(*
Geographic Pose
----------------

Overview
================
Represents a coordinate system on a reference ellipsoid.
Similar to the HMatrix transformation, but based on an ellipsoid instead of in cartesian space (helper functions are included to switch between HMatrix and GeoPose).
Represents the geodetic (or geocentric) position with latitude, longitude, and elevation (above the ellipsoid) - Accessed with the 'Position' property.
Represents the orientation as a set of angles relative to the ENU tangent coordinate system at the CS origin - Accessed with the 'Orientation' property.
*)
FUNCTION_BLOCK GeoPose
VAR_INPUT
END_VAR
VAR_OUTPUT
END_VAR
VAR
	Position_ : GeoPosition;//ECEF
	Orientation_ : TaitBryanAngleOrientation;//ENU at position
END_VAR

METHOD PUBLIC Clear
VAR_INPUT
END_VAR
Position_.Clear();
Orientation_.Clear();
END_METHOD

METHOD PUBLIC CopyFrom
VAR_INPUT
	P : GeoPose;
END_VAR
Position_.CopyFrom(P.Position_);
Orientation_.CopyFrom(P.Orientation_);
END_METHOD

METHOD PUBLIC GetEcefTransformation : HMatrix
VAR_INPUT
	Ref : REFERENCE TO GeoEllipsoid := GeoEllipsoids.WGS84;
END_VAR
VAR
	EnuInEcef : HMatrix;//holds the geoposition part, and the tangent rotation
	ThisInEnu : HMatrix;//just holds the local rotation portion
END_VAR
EnuInEcef := Position_.GetTangentEnuTransform(Ref);
ThisInEnu.RMatrixComponent := Orientation_.GetRMatrix();
GetEcefTransformation := EnuInEcef.GetTransformedHMatrix(ThisInEnu);
END_METHOD

METHOD PUBLIC GetRelativeOrientation : TaitBryanAngleOrientation
VAR_INPUT
	P : GeoPose;
	Ref : REFERENCE TO GeoEllipsoid := GeoEllipsoids.WGS84;
END_VAR
VAR
	ThisInEcef : HMatrix;
	InputInThis : HMatrix;
END_VAR
ThisInEcef := GetEcefTransformation(Ref);
InputInThis := ThisInEcef.GetTransformedHMatrixReverse(P.GetEcefTransformation(Ref));
GetRelativeOrientation.SetFromRMatrix(InputInThis.RMatrixComponent);
END_METHOD

METHOD PUBLIC GetRelativePosition : Vector3
VAR_INPUT
	P : GeoPose;
	Ref : REFERENCE TO GeoEllipsoid := GeoEllipsoids.WGS84;
END_VAR
VAR
	ThisInEcef : HMatrix;
	InputInThis : HMatrix;
END_VAR
ThisInEcef := GetEcefTransformation(Ref);
InputInThis := ThisInEcef.GetTransformedHMatrixReverse(P.GetEcefTransformation(Ref));
GetRelativePosition := InputInThis.Vector3Component;
END_METHOD

METHOD PUBLIC IsEqual : BOOL
VAR_INPUT
	P : GeoPose;
END_VAR
IsEqual := IsNearlyEqual(P,0.0,0.0,0.0);
END_METHOD

METHOD PUBLIC IsNearlyEqual : BOOL
VAR_INPUT
	P : GeoPose;
	PositionPrecisionLatLon : LREAL;//rad
	PositionPrecisionElevation : LREAL;//m
	OrientationPrecision : LREAL;//radians
END_VAR
IsNearlyEqual := Position_.IsNearlyEqual(P.Position_, PositionPrecisionLatLon, PositionPrecisionElevation) AND Orientation_.IsNearlyEqual(P.Orientation_, OrientationPrecision);
END_METHOD

PROPERTY PUBLIC Orientation : TaitBryanAngleOrientation
GET
Orientation.CopyFrom(Orientation_);
END_GET
SET
Orientation_.CopyFrom(Orientation);
END_SET
END_PROPERTY

PROPERTY PUBLIC Position : GeoPosition
GET
Position.CopyFrom(Position_);
END_GET
SET
Position_.CopyFrom(Position);
END_SET
END_PROPERTY

METHOD PUBLIC SetFromComponents
VAR_INPUT
	P : GeoPosition;
	O : TaitBryanAngleOrientation;
END_VAR
Position_.CopyFrom(P);
Orientation_.CopyFrom(O);
END_METHOD

METHOD PUBLIC SetFromEcefTransformation
VAR_INPUT
	H : HMatrix;//ThisInEcef)
	Ref : REFERENCE TO GeoEllipsoid := GeoEllipsoids.WGS84;
END_VAR
VAR
	EnuInEcef : HMatrix;
	ThisInEnu : HMatrix;
END_VAR
Clear();
Position_.SetFromCartesianPosition(H.Vector3Component,Ref);
EnuInEcef := Position_.GetTangentEnuTransform(Ref);
ThisInEnu := EnuInEcef.GetTransformedHMatrixReverse(H);
Orientation_.SetFromRMatrix(ThisInEnu.RMatrixComponent);
END_METHOD

END_FUNCTION_BLOCK

(* stored: Version 1.1.0.1, ProductVersion 3.1.4024.9
   POU GeoPose: Id {22fd7b91-e379-4b48-b25b-7c3f882da5ab}, SpecialFunc None
   Folder Comparators: Id {128afaf1-84d6-4df8-a22c-9d3f4b4940a4}
   Folder Helpers: Id {67e259ad-2bdb-48bf-a64f-ac35164c5381}
   Folder Properties: Id {997fd598-578a-47c3-a5a0-4cda164034ca}
   Folder Setters: Id {56adf730-714f-4820-85ec-55dba9a85f39}
   Method Clear: Id {ac1dee2d-66a0-48f3-805d-a8a5da1d833f}
   Method CopyFrom: Id {dba523a8-541c-484d-aa76-3d7ae4f213a4}
   Method GetEcefTransformation: Id {e681c242-06fb-4148-88fe-37c56511e90a}
   Method GetRelativeOrientation: Id {d190558d-a28b-485d-a2dd-6e0e06e2ef1c}
   Method GetRelativePosition: Id {7569a23a-af29-4f3c-a02f-18ac30d21f8f}
   Method IsEqual: Id {407842f3-df1e-4c43-b83b-80af1e674f13}
   Method IsNearlyEqual: Id {d4e7d56a-e971-4ba6-989b-27514f27105d}
   Property Orientation: Id {1d991835-c59d-472a-9f50-c2009c261e0f}
   Get Get: Id {08d8e7ad-d8cc-4d59-93fd-4c65600b7bf3}
   Set Set: Id {50610a45-4344-45ff-a9d7-6a21cdf93b88}
   Property Position: Id {97c7942e-3eae-40dd-8bd3-b21545263991}
   Get Get: Id {2021bfe0-3706-444f-b949-eb89d2296220}
   Set Set: Id {5cf0345f-1fc2-4982-8bb0-50d9afb0185e}
   Method SetFromComponents: Id {f2babd1a-506a-402c-9541-fa8625b67834}
   Method SetFromEcefTransformation: Id {3f187cfe-7854-444b-8e8e-cef8b71a29c5} *)
